// TIA Portal V20 export
DATA_BLOCK "HMI_SideShifter_2"   // DB41
{ S7_Optimized_Access := 'TRUE' }
// stored: MemoryReserve 100
   VAR
      SL_Go_Forward : Bool;
      SL_Go_Backward : Bool;
      SL_Velocity : Int;
      SL_Hydraulic_Unit : Bool;
      SL_Actuators_Push : Bool;
      SL_Actuators_Pull : Bool;
      Go_to_ST25 : Bool;
      Go_to_ST24 : Bool;
      Go_to_ST17 : Bool;
      Go_to_ST14 : Bool;
      SR_SL_Hyd_Up : Bool;
      SR_SL_Hyd_Down : Bool;
      SR_Go_Forward : Bool;
      SR_Go_Backward : Bool;
      SR_Velocity : Int;
      SR_Hydraulic_Unit : Bool;
      SR_Actuators_Push : Bool;
      SR_Actuators_Pull : Bool;
      Reset_Drives : Bool;
      Reset_Hydro : Bool;
   END_VAR
   VAR RETAIN
      Homing_SL1 : Int := 1860;
      Homing_SL2 : Int := 7461;
      Homing_SL3 : Int := 13450;
      Homing_SL4 : Int := 19048;
      Homing_SR1 : Int := 1868;
      Homing_SR2 : Int := 7469;
      Homing_SR3 : Int := 13465;
      Homing_SR4 : Int := 19056;
   END_VAR
BEGIN
END_DATA_BLOCK
